PROGRAM MAIN
VAR
	M1 : DUT_MotionStage:=(nCOmmand:=3); // Bender Motor
	fbMotionStage : FB_MotionStage;
	bSTOEnable AT %I* : BOOL;
END_VAR

// Button to enable motor: write 0 to enable, 2 to disable
M1.nEnableMode;

// Tie STO into Enable Bit:
M1.bHardwareEnable := bSTOEnable;

// Start Motion
fbMotionStage (stMotionStage:=M1);

END_PROGRAM

(* stored: Version 1.1.0.1, ProductVersion 3.1.4022.18
   POU MAIN: Id {2f9042fa-41a7-4fd2-8aa4-dee837e83b8e}, SpecialFunc None *)
